FUNCTION_BLOCK FB_TrackSegment_2 EXTENDS FB_TrackBase IMPLEMENTS I_TRACK
VAR_INPUT
END_VAR
VAR_OUTPUT
END_VAR

METHOD Initialize : BOOL

VAR_INPUT
	nTrackIndex : UDINT;
END_VAR


VAR_INST
	TrackTable		: FB_TrackTable;
	
	nPointIndex		: INT;
	nPointIndexA	: INT;	
	nPointIndexB	: INT;	
	idx1, idx2		: INT;
	nStartFromTrack	: INT;
	nEndAtTrack		: INT;
	bCloseLoop		: BOOL;	
	
	bTrackBuild		: BOOL;
	StartFromTrack	: I_Track;
	EndAtTrack		: I_Track;
	
	sIndexWhereTheCheckFailed	: UINT;
	nErrorID					: UDINT;

END_VAR





VAR_INST
	
	TrackTableTemp		: ARRAY[1..gc_MaxNumberTrackPoints] OF ST_TrackTable;
	


END_VAR


VAR_INST
	
	pos01	:		PositionXYC;
	pos02	:		PositionXYC;


END_VAR

	  
CASE nState OF 

	10:	// Starting with an empty table. 
		IF TrackTable.ClearTrackTable() THEN
			nState := nState + 10;
		END_IF
		

	20:	// Init Track-Table
		
		// *************************************************************************************
		// *** Only the code in this state must be eddited according to machine/track layout ***
		// *************************************************************************************	
		
		nStartFromTrack	:= 1;		// 0 for the first track all others according to their predecessor!
	    	nEndAtTrack := 1;		// 0 for the first track all others according to their successor! 		
		     bCloseLoop := FALSE;	// TRUE for circular track	

			 			 			 
		// Building the track table:
		TrackTable.AddPoint(E_PointType.Line_Start, E_PointOption.none, 600.0, 480.0, 0.0); 	 
		TrackTable.AddPoint(E_PointType.Line_End,   E_PointOption.none, 600.0, 240.0, 0.0);				
						
		nState := nState + 10;


	30:
		// *************************************************************
		// ***       NO Code Changes are needed from here on!        ***
		// *************************************************************		
			
		// The track table contains all additional information, too.
		IF nStartFromTrack > 0 THEN
			TrackTable.P_StartFromTrack := ipTrack[nStartFromTrack].std;	
		END_IF
		IF nEndAtTrack > 0 THEN
			TrackTable.P_EndAtTrack := ipTrack[nEndAtTrack].std;	
		END_IF	
		TrackTable.P_CloseTheLoop := bCloseLoop;	
		nState := nState + 10;

			
		
	40: // Checking the track table for plausibility
		IF TrackTable.CheckTrackTable() <> 0 THEN
			IF TrackTable.P_TrackTableCheckResult THEN
				nState := 50;	// Plausibility test succeeded.
			ELSE
				nState := 41;	// Plausibility test failed!
			END_IF
		END_IF

	
	41:	// In case of failed plausibility test check the creation of the above track table.
		// A Line must always begin with E_PointType.Line_Start and end with E_PointType.Line_End.
		// A Circle must always be added in the order E_PointType.Circle_Start, E_PointType.Circle_Center, E_PointType.Circle_End.
		// Check the info text for further information:
		sErrorInfoTextTemp := CONCAT('Track: ', UDINT_TO_STRING(nTrackIndex));
		sErrorInfoTextTemp := CONCAT(sErrorInfoTextTemp, ' - ');
		sErrorInfoTextTemp := CONCAT(sErrorInfoTextTemp, TrackTable.P_InfoText);
		
				     bTrackBuildError := TRUE;
					   sErrorInfoText := sErrorInfoTextTemp;
			sIndexWhereTheCheckFailed := TrackTable.P_TrackCheckImplausibleTableIndex;
					   TrackTableTemp := TrackTable.P_Table;	
							
 					   
	50:	// Building the track	
		IF fbTrackStandard.BuildTrackExt(TrackTable) THEN
			nState := nState +1;
		END_IF
		
	51:	IF fbTrackStandard.P_BuildTrackExt.Done THEN
			nState := 100;	
		ELSIF fbTrackStandard.P_BuildTrackExt.Error THEN
	  		nState := nState +1;
		END_IF		
		
	52: // In case an error occured, check the error ID and InfoText and react accordingly:
		sErrorInfoTextTemp := CONCAT('Track: ', UDINT_TO_STRING(nTrackIndex));
		sErrorInfoTextTemp := CONCAT(sErrorInfoTextTemp, ' - ');
		sErrorInfoTextTemp := CONCAT(sErrorInfoTextTemp, fbTrackStandard.P_BuildTrackExtInfoText);	
	
			      nErrorID := fbTrackStandard.P_BuildTrackExt.ErrorID;
		    sErrorInfoText := sErrorInfoTextTemp;		
			
		  bTrackBuildError := TRUE;		   
					   
		 
	100: 	// Track build done
			fTrackLength := fbTrackStandard.GetLength();
			  Initialize := TRUE;
	
			
END_CASE
END_METHOD

PROPERTY P_Error : BOOL
GET
P_Error := bTrackBuildError;
END_GET
END_PROPERTY

PROPERTY P_ErrorInfo : STRING
GET
P_ErrorInfo := sErrorInfoText;
END_GET
END_PROPERTY

END_FUNCTION_BLOCK

(* stored: Version 1.1.0.1, ProductVersion 3.1.4024.13
   POU FB_TrackSegment_2: Id {9802caed-2bc3-40a6-bd4e-7f09158977a4}, SpecialFunc None
   Method Initialize: Id {6b9a48cc-fd1e-4477-abf8-bc24a07575aa}
   Property P_Error: Id {134d47f6-3f43-4dbc-8f80-60528b3bb860}
   Get Get: Id {43084986-85d7-418e-96e3-a3f0310f7c8b}
   Property P_ErrorInfo: Id {d2173afd-4b82-4137-92b4-366957b7a143}
   Get Get: Id {a31c5326-cf7e-473a-ac1b-a6f9e3b894cc} *)
